Fanuc KAREL source: kt00128.KL

-- PROVISIONAL review KL for V770-1; original PC SHA256 8ed54c82454b697897cfd92b2ebd4cf7bb90ea7bd3b7d4bc1a4c284b1a5f19df
-- Incomplete behavior may be omitted. Consult companion uncertainty JSON. Do not deploy.
PROGRAM KT00128
%NOLOCKGROUP
VAR
  OUT : REAL
-- UNRESOLVED_DECL H1 type=002017
-- UNRESOLVED_DECL H2 type=002017
BEGIN
  -- UNRESOLVED_PC offsets 5-19; opcodes 2E,22,9D,33,B4
  -- UNRESOLVED_PC offsets 24-38; opcodes 2E,22,9D,33,B4
  -- UNRESOLVED_PC offsets 43-57; opcodes 2E,22,9D,33,B4
  -- UNRESOLVED_PC offsets 62-76; opcodes 2E,22,9D,33,B4
  -- UNRESOLVED_PC offsets 81-110; opcodes 22,9D,33,B3,22,9D,33,B3,64,29,64,29,6C,23
  -- UNRESOLVED_PC offsets 115-119; opcodes 7F
END KT00128
